// TIA Portal V18 export
FUNCTION_BLOCK "man_descrete_sr"   // FB28, FBD
{ S7_Optimized_Access := 'TRUE' }
VERSION : 0.1
// stored: AutoNumber true, IsIECCheckEnabled false, IsRetainMemResEnabled false, MemoryReserve 100, SetENOAutomatically false, UDAEnableTagReadback false
   VAR_INPUT
      condions : Bool;
      buttons : Bool;
      arrived : Bool;
   END_VAR
   VAR_OUTPUT
      exce_man : Bool;
   END_VAR
BEGIN

REGION Network 1
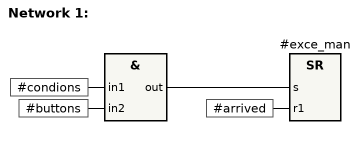
   IF #condions AND #buttons THEN
       #exce_man := TRUE;   // SR flip-flop
   END_IF;
   IF #arrived THEN #exce_man := FALSE; END_IF;
END_REGION
END_FUNCTION_BLOCK
